TYPE DUT_STRUCT_VARIABLES :
STRUCT
	sEnvironment		:STRING;
	sCellName			:STRING;
	sIpAddress			:STRING;
	sAmsNetId			:STRING;
	sOpcUaURL			:STRING;
//	sUhfRfidOpcUaURL	:STRING;
//	sHfRfidOpcUaURL		:STRING;
	sStation1			:STRING;
	sTrackserver		:STRING;
	sTrackserver_AMS	:STRING;
//	sStation2			:STRING;
//	sStation3			:STRING;
//	sStation4			:STRING;
//	sRelease			:STRING;
//	sCommitID			:STRING;
//	sTag				:STRING;
END_STRUCT
END_TYPE

(* stored: Version 1.1.0.1, ProductVersion 3.1.4024.5
   DUT DUT_STRUCT_VARIABLES: Id {75fee008-bd74-4965-a6e1-e2126a79bf49} *)
